(* generate basic date time format with no dashes*)
FUNCTION F_SYSTEM_SystemTimeToOHMFolderName : STRING(33)
VAR_INPUT
	sSystemTime			: TIMESTRUCT;
END_VAR
VAR
	strYear				: STRING(4);
	strMonth				: STRING(2);
	strDay				: STRING(2);

	strDate				: STRING(10);
END_VAR

(*Date*)
	strYear:=F_StringAddPrefix(WORD_TO_STRING(sSystemTime.wYear), 4, '0');
	strMonth:=F_StringAddPrefix(WORD_TO_STRING(sSystemTime.wMonth), 2, '0');
	strDay:=F_StringAddPrefix(WORD_TO_STRING(sSystemTime.wDay), 2, '0');

(*Print*)
	strDate := F_CONCAT3(strYear, strMonth, strDay);
	F_SYSTEM_SystemTimeToOHMFolderName := strDate;

END_FUNCTION

(* stored: Version 1.1.0.1, ProductVersion 3.1.4024.15
   POU F_SYSTEM_SystemTimeToOHMFolderName: Id {b397e41f-3082-45b6-8487-b05dfd7c4106}, SpecialFunc None *)
